ABB RobotStudio station: Lab1_HW_Jozefovic_217281.rspag

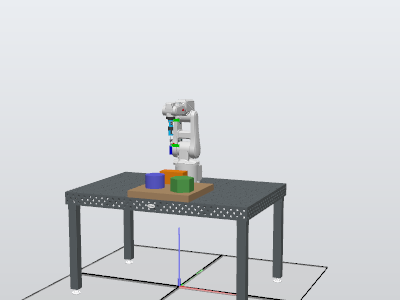
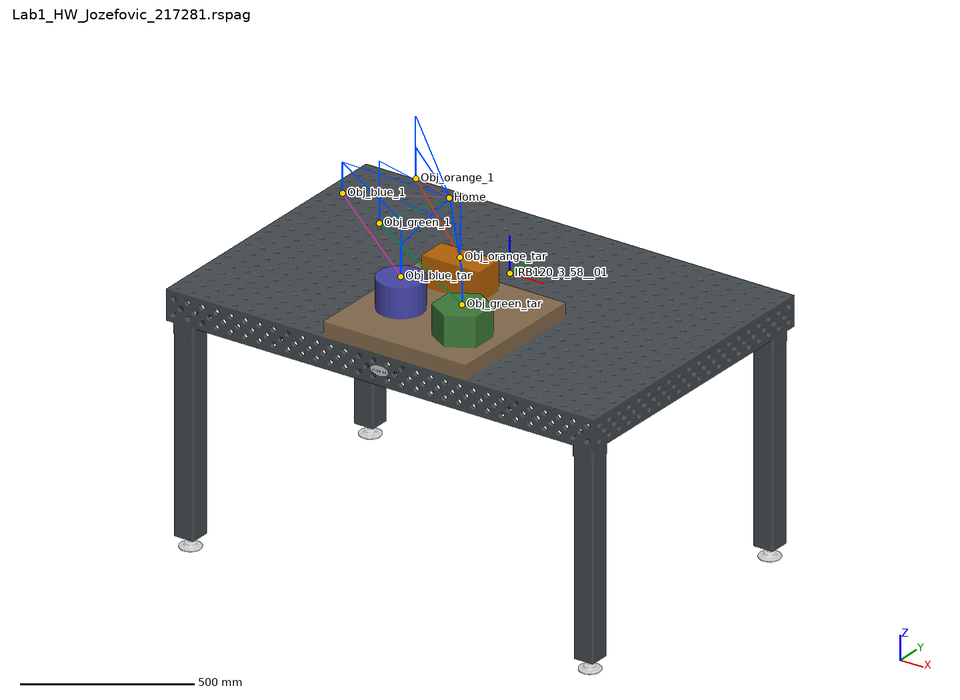
[picture v1: parts stored in the station drawn from their meshes, with robot base, taught points and paths (robot models come from the ABB library and are not in the file)]
--- station ---
Station Solution_1_Tutorial (saved by RobotStudio 22.3.10190.2)
Controller Controller1, task T_ROB1: task frame (RAPID world) sits at (0, 150, 830) mm, rotated rx 0 ry 0 rz -90 deg in the station
Controller Controller1
  mechanical unit ROB_1: IRB120_3_58__01, 6 joints, base frame (0, 0, 0) mm
Layout (positions relative to the parent item):
  - table [part] at (-200, -500, 830) mm, size 500 x 500 x 50 mm
  - object_1 [part] at (-200, -500, 830) mm, size 200 x 100 x 150 mm
  - object_2 [part] at (-200, -500, 829.99) mm, size 149.5 x 149.7 x 150 mm
  - object_3 [part] at (-200, -500, 830) mm, size 155.5 x 179.5 x 150 mm
  - siegmund_1500_1000 [part], size 1500 x 1010.3 x 830 mm
  - object_11 [part] at (-200, -500, 830) mm, size 200 x 100 x 150 mm
  - object_22 [part] at (-200, -500, 830) mm, size 149.5 x 149.7 x 150 mm
  - object_33 [part] at (-200, -500, 830) mm, size 155.5 x 179.5 x 150 mm
  - IRB120_3_58__01 [mechanism, from Robots\IRB120_3_58_G_01.rslib] at (0, 150, 830) mm, rotated rx 0 ry 0 rz -90 deg; joint values [0, 0, 0, 0, 1.5708, 0] (rad or m)
  - smc_gripper [mechanism, from Gripper_RS_tool\smc_gripper.rslib] at (0, -152, 1388) mm, rotated rx 180 ry 0 rz 90 deg
  - Positioner [smart component, from Components\Positioner.rslib]
      properties: Object=object_1; Position=[-0.6 -0.15 0.83]; Orientation=[0 0 0]; Reference=Global; ReferenceObject=(none)
  - Attacher [smart component, from Components\Attacher.rslib]
      properties: Parent=smc_gripper; Flange=0; Child=object_1; Mount=false; Offset=[0 0 0]; Orientation=[0 0 0]
  - Detacher [smart component, from Components\Detacher.rslib]
      properties: Child=object_1; KeepPosition=true
  - Attacher_2 [smart component, from Components\Attacher.rslib]
      properties: Parent=smc_gripper; Flange=0; Child=object_3; Mount=false; Offset=[0 0 0]; Orientation=[0 0 0]
  - Detacher_2 [smart component, from Components\Detacher.rslib]
      properties: Child=object_3; KeepPosition=true
  - Attacher_3 [smart component, from Components\Attacher.rslib]
      properties: Parent=smc_gripper; Flange=0; Child=object_2; Mount=false; Offset=[0 0 0]; Orientation=[0 0 0]
  - Detacher_4 [smart component, from Components\Detacher.rslib]
      properties: Child=object_2; KeepPosition=true
  - Positioner_3 [smart component, from Components\Positioner.rslib]
      properties: Object=object_3; Position=[-0.7 -0.2 0.83]; Orientation=[0 0 0]; Reference=Global; ReferenceObject=(none)
  - Positioner_4 [smart component, from Components\Positioner.rslib]
      properties: Object=object_2; Position=[-0.65 -0.15 0.83]; Orientation=[0 0 0]; Reference=Global; ReferenceObject=(none)
Attachment: smc_gripper is attached to IRB120_3_58__01 / Link6
Collision set CollisionSet_1: object_1 against object_2, object_3, near miss 0 m
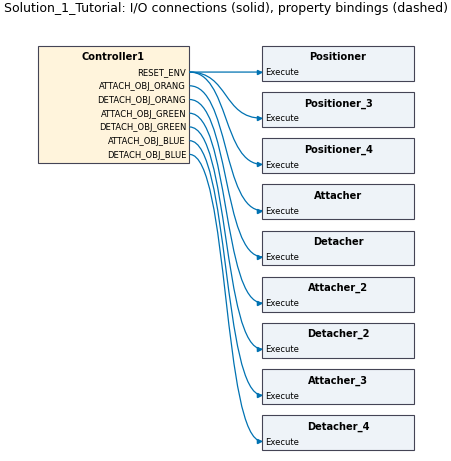
Station logic (signal -> signal, property => property):
  Controller1.RESET_ENV -> Positioner.Execute
  Controller1.ATTACH_OBJ_ORANGE -> Attacher.Execute
  Controller1.DETACH_OBJ_ORANGE -> Detacher.Execute
  Controller1.ATTACH_OBJ_GREEN -> Attacher_2.Execute
  Controller1.DETACH_OBJ_GREEN -> Detacher_2.Execute
  Controller1.ATTACH_OBJ_BLUE -> Attacher_3.Execute
  Controller1.DETACH_OBJ_BLUE -> Detacher_4.Execute
  Controller1.RESET_ENV -> Positioner_3.Execute
  Controller1.RESET_ENV -> Positioner_4.Execute

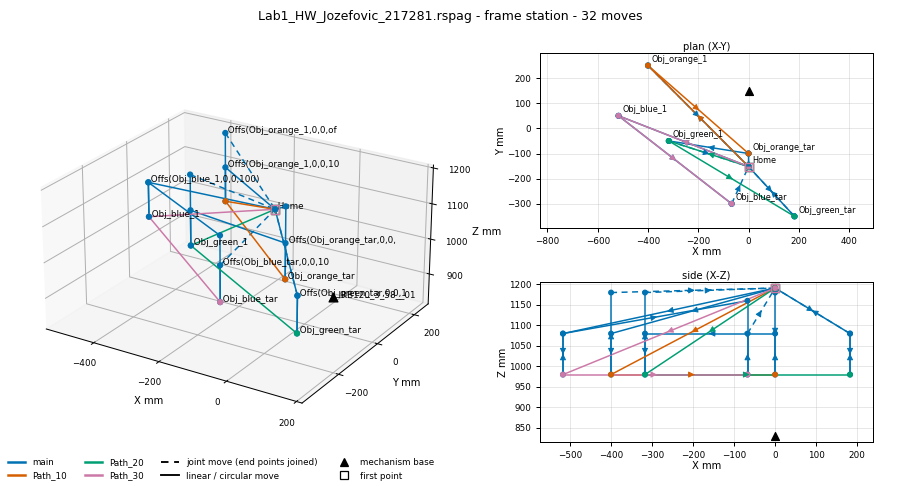
[picture p0: tool path of Lab1_HW_Jozefovic_217281.rspag in frame station, 32 of 32 moves have a stored position in this frame; points joined in program order, loops and branches not executed]
--- Backups/Controller1/RAPID/TASK1/PROGMOD/CalibData.mod ---
MODULE CalibData
    PERS tooldata smc_gripper:=[TRUE,[[0,0.004,197.001],[1,0,0,0]],[1,[0.207,-0.496,71.18],[1,0,0,0],0,0,0]];
ENDMODULE

--- Backups/Controller1/RAPID/TASK1/PROGMOD/Module1.mod ---
MODULE Module1
    CONST robtarget Home:=[[302,0.004,360.999],[0,0,1,0],[-1,0,-1,0],[9E+09,9E+09,9E+09,9E+09,9E+09,9E+09]];
    !ORANGE
    CONST robtarget Obj_orange_1:=[[-100,-400,150],[0,0,1,0],[-2,0,-2,0],[9E+09,9E+09,9E+09,9E+09,9E+09,9E+09]];
    CONST robtarget Obj_orange_tar:=[[250,0,150],[0,0,1,0],[-1,0,-1,0],[9E+09,9E+09,9E+09,9E+09,9E+09,9E+09]];
    !GREEN
    CONST robtarget Obj_green_1:=[[200,-317.298,150],[0,0,1,0],[-1,0,-1,0],[9E+09,9E+09,9E+09,9E+09,9E+09,9E+09]];
    CONST robtarget Obj_green_tar:=[[500,182.702,150],[0,0,1,0],[0,0,0,0],[9E+09,9E+09,9E+09,9E+09,9E+09,9E+09]];
    !BLUE
    CONST robtarget Obj_blue_1:=[[100,-517.298,150],[0,0,1,0],[-1,0,-1,0],[9E+09,9E+09,9E+09,9E+09,9E+09,9E+09]];
    CONST robtarget Obj_blue_tar:=[[450,-67.298,150],[0,0,1,0],[0,0,0,0],[9E+09,9E+09,9E+09,9E+09,9E+09,9E+09]];

    VAR num offset_z := 200;

    PROC main()
        !Reset env
        PulseDO DETACH_OBJ_ORANGE;
        PulseDO DETACH_OBJ_BLUE;
        PulseDO DETACH_OBJ_GREEN;
        PulseDO RESET_ENV;

        !Home posi
        MoveJ Home,v800,fine,smc_gripper\WObj:=wobj0;

        !MoveL Obj_orange_1,v100,fine,smc_gripper\WObj:=wobj0;
        !Pick obj orange
        MoveL Offs(Obj_orange_1,0,0,100),v600,z50,smc_gripper\WObj:=wobj0;
        MoveL Offs(Obj_orange_1,0,0,0),v400,fine,smc_gripper\WObj:=wobj0;
            !Attaching
        PulseDO ATTACH_OBJ_ORANGE;
        WaitTime 0.6;
        MoveL Offs(Obj_orange_1,0,0,offset_z),v200,z50,smc_gripper\WObj:=wobj0;

        !Home posi
        MoveJ Home,v200,z100,smc_gripper\WObj:=wobj0;

        !place obj orange
        MoveL Offs(Obj_orange_tar,0,0,offset_z),v200,z50,smc_gripper\WObj:=wobj0;
        MoveL Offs(Obj_orange_tar,0,0,0),v200,fine,smc_gripper\WObj:=wobj0;
            !Detaching
        PulseDO DETACH_OBJ_ORANGE;
        WaitTime 0.4;
        MoveL Offs(Obj_orange_tar,0,0,100),v400,z50,smc_gripper\WObj:=wobj0;

        !Home posi

        !-------GREEN GREEN GREEN GREEN GREEN GREEN-----------

        !Pick obj green
        MoveL Offs(Obj_green_1,0,0,100),v600,z50,smc_gripper\WObj:=wobj0;
        MoveL Offs(Obj_green_1,0,0,0),v400,fine,smc_gripper\WObj:=wobj0;
            !Attaching
        PulseDO ATTACH_OBJ_GREEN;
        WaitTime 0.6;
        MoveL Offs(Obj_green_1,0,0,offset_z),v200,z50,smc_gripper\WObj:=wobj0;

        !Home posi
        MoveJ Home,v200,z100,smc_gripper\WObj:=wobj0;

        !place obj orange
        MoveL Offs(Obj_green_tar,0,0,100),v200,z100,smc_gripper\WObj:=wobj0;
        MoveL Offs(Obj_green_tar,0,0,0),v200,fine,smc_gripper\WObj:=wobj0;
            !Detaching
        PulseDO DETACH_OBJ_GREEN;
        WaitTime 0.4;
        MoveL Offs(Obj_green_tar,0,0,100),v400,z50,smc_gripper\WObj:=wobj0;

        !Home posi
        MoveJ Home,v600,z100,smc_gripper\WObj:=wobj0;

        !-------BLUE BLUE BLUE BLUE BLUE BLUE BLUE BLUE-----------

        !Pick obj blue
        MoveL Offs(Obj_blue_1,0,0,100),v600,z50,smc_gripper\WObj:=wobj0;
        MoveL Offs(Obj_blue_1,0,0,0),v400,fine,smc_gripper\WObj:=wobj0;
            !Attaching
        PulseDO ATTACH_OBJ_BLUE;
        WaitTime 0.6;
        MoveL Offs(Obj_blue_1,0,0,100),v200,z50,smc_gripper\WObj:=wobj0;

        !place obj blue
        MoveL Offs(Obj_blue_tar,0,0,180),v200,z50,smc_gripper\WObj:=wobj0;
        MoveL Offs(Obj_blue_tar,0,0,0),v200,fine,smc_gripper\WObj:=wobj0;
            !Detaching
        PulseDO DETACH_OBJ_BLUE;
        WaitTime 0.4;
        MoveL Offs(Obj_blue_tar,0,0,100),v400,z50,smc_gripper\WObj:=wobj0;

        !Home posi
        MoveJ Home,v600,fine,smc_gripper\WObj:=wobj0;

    ENDPROC

    PROC Path_10()
        MoveL Home,v100,fine,smc_gripper\WObj:=wobj0;
        MoveL Obj_orange_1,v100,fine,smc_gripper\WObj:=wobj0;
        MoveL Obj_orange_tar,v100,fine,smc_gripper\WObj:=wobj0;
    ENDPROC
    PROC Path_20()
        MoveL Home,v1000,z100,smc_gripper\WObj:=wobj0;
        MoveL Obj_green_1,v1000,z100,smc_gripper\WObj:=wobj0;
        MoveL Obj_green_tar,v1000,z100,smc_gripper\WObj:=wobj0;
    ENDPROC
    PROC Path_30()
        MoveL Home,v1000,z100,smc_gripper\WObj:=wobj0;
        MoveL Obj_blue_1,v1000,z100,smc_gripper\WObj:=wobj0;
        MoveL Obj_blue_tar,v1000,z100,smc_gripper\WObj:=wobj0;
    ENDPROC
ENDMODULE

--- Backups/Controller1/SYSPAR/EIO.cfg ---
EIO:CFG_1.0:6:1::
#
EIO_SIGNAL:

      -Name "RESET_ENV" -SignalType "DO"

      -Name "ATTACH_OBJ_ORANGE" -SignalType "DO"

      -Name "DETACH_OBJ_ORANGE" -SignalType "DO"

      -Name "ATTACH_OBJ_GREEN" -SignalType "DO"

      -Name "ATTACH_OBJ_BLUE" -SignalType "DO"

      -Name "DETACH_OBJ_GREEN" -SignalType "DO"

      -Name "DETACH_OBJ_BLUE" -SignalType "DO"
